FUNCTION plusOuMoins : bool
VAR_INPUT
	val1  : LREAL;
	val2  : LREAL;
	plage : LREAL;
END_VAR

IF val1 < val2 + plage AND val1 > val2 - plage THEN 
	plusOuMoins := TRUE;
ELSE
	plusOuMoins := FALSE;
END_IF

END_FUNCTION

(* stored: Version 1.1.0.1, ProductVersion 3.1.4024.11
   POU plusOuMoins: Id {985b8a85-c5bf-4959-87a2-f54d0b76c8df}, SpecialFunc None *)
